TYPE ST_HallAssignment :
STRUCT
	posDirection: BOOL;
	nTripCount: INT;
	calNseq: WORD;
	eventNseq: WORD;
	calEdge: BOOL;
	eventEdge: BOOL;
	calPos: LREAL;
	goNextSeq: BOOL;
END_STRUCT
END_TYPE

(* stored: Version 1.1.0.1, ProductVersion 3.1.4022.18
   DUT ST_HallAssignment: Id {cdc908b1-35d7-43f1-ae6b-4ea7a1693955} *)
